{attribute 'qualified_only'}
VAR_GLOBAL CONSTANT
    nModule : SINT := 1;
END_VAR

(* stored: Version 1.1.0.1
   GVL nBundleStages: Id {0c986dc4-1677-483e-a0bf-f21be608e84f}, ParameterList True *)
